TEXTLIST TextList
  1 = 'testun' | EN: 'Testone' | FR: 'Testun'
   = ''
END_TEXTLIST

(* stored: Version 1.1.0.1
   TextList TextList: Id {d373a37d-c7ea-4948-adb6-7854078e3b40} *)
